// Mitsubishi GX Works2 project: BookEX6_42 DataControl   PLC: Q13UDV

// global labels: Global
VAR_GLOBAL
  bVar0 AT M5000 : BOOL;
  abArray0 AT M5010 : ARRAY [0..49] OF BOOL;
  sStr0 AT D5000 : STRING[199];
  sStr1 AT D5100 : STRING[199];
  sStr2 AT D5200 : STRING[199];
  sStr3 AT D5300 : STRING[199];
  sStr4 AT D5400 : STRING[199];
  sStr5 AT D5500 : STRING[199];
  sStr6 AT D5600 : STRING[199];
  sStr7 AT D5700 : STRING[199];
  sStr8 AT D5800 : STRING[199];
  sStr9 AT D5900 : STRING[199];
  iVar0 AT D4500 : INT;
  iVar1 AT D4501 : INT;
  iVar2 AT D4502 : INT;
  iVar3 AT D4503 : INT;
  iVar4 AT D4504 : INT;
  iVar5 AT D4505 : INT;
  iVar6 AT D4506 : INT;
  iVar7 AT D4507 : INT;
  iVar8 AT D4508 : INT;
  iVar9 AT D4509 : INT;
  dVar0 AT D4510 : DINT;
  dVar1 AT D4512 : DINT;
  dVar2 AT D4514 : DINT;
  dVar3 AT D4516 : DINT;
  dVar4 AT D4518 : DINT;
  dVar5 AT D4520 : DINT;
  dVar6 AT D4522 : DINT;
  dVar7 AT D4524 : DINT;
  dVar8 AT D4526 : DINT;
  dVar9 AT D4528 : DINT;
  wVar0 AT D4530 : WORD;
  wVar1 AT D4531 : WORD;
  wVar2 AT D4532 : WORD;
  wVar3 AT D4533 : WORD;
  wVar4 AT D4534 : WORD;
  wVar5 AT D4535 : WORD;
  wVar6 AT D4536 : WORD;
  wVar7 AT D4537 : WORD;
  wVar8 AT D4538 : WORD;
  wVar9 AT D4539 : WORD;
  dwVar0 AT D4540 : DWORD;
  dwVar1 AT D4542 : DWORD;
  dwVar2 AT D4544 : DWORD;
  dwVar3 AT D4546 : DWORD;
  dwVar4 AT D4548 : DWORD;
  dwVar5 AT D4550 : DWORD;
  dwVar6 AT D4552 : DWORD;
  dwVar7 AT D4554 : DWORD;
  dwVar8 AT D4556 : DWORD;
  dwVar9 AT D4558 : DWORD;
  fsVar0 AT D4560 : REAL;
  fsVar1 AT D4562 : REAL;
  fsVar2 AT D4564 : REAL;
  fsVar3 AT D4566 : REAL;
  fsVar4 AT D4568 : REAL;
  fsVar5 AT D4570 : REAL;
  fsVar6 AT D4572 : REAL;
  fsVar7 AT D4574 : REAL;
  fsVar8 AT D4576 : REAL;
  fsVar9 AT D4578 : REAL;
  fdVar0 AT D4580 : LREAL;
  tTime0 AT D4620 : TIME;
  tTime1 AT D4622 : TIME;
  tTime2 AT D4624 : TIME;
  tTime3 AT D4626 : TIME;
  tTime4 AT D4628 : TIME;
  tTime5 AT D4630 : TIME;
  tTime6 AT D4632 : TIME;
  tTime7 AT D4634 : TIME;
  tTime8 AT D4636 : TIME;
  tTime9 AT D4638 : TIME;
  tTime10 AT D4640 : TIME;
  bVar1 AT M5001 : BOOL;
  bVar2 AT M5002 : BOOL;
  bVar3 AT M5003 : BOOL;
  bVar4 AT M5004 : BOOL;
  bVar5 AT M5005 : BOOL;
  bVar6 AT M5006 : BOOL;
  bVar7 AT M5007 : BOOL;
  bVar8 AT M5008 : BOOL;
  bVar9 AT M5009 : BOOL;
  abArray1 AT M5060 : ARRAY [0..49] OF BOOL;
  abArray2 AT M5110 : ARRAY [0..49] OF BOOL;
  abArray3 AT M5160 : ARRAY [0..49] OF BOOL;
  abArray4 AT M5210 : ARRAY [0..49] OF BOOL;
  abArray5 AT M5260 : ARRAY [0..49] OF BOOL;
  abArray6 AT M5310 : ARRAY [0..49] OF BOOL;
  abArray7 AT M5360 : ARRAY [0..49] OF BOOL;
  abArray8 AT M5410 : ARRAY [0..49] OF BOOL;
  abArray9 AT M5460 : ARRAY [0..49] OF BOOL;
  fdVar1 AT D4584 : LREAL;
  fdVar2 AT D4588 : LREAL;
  fdVar3 AT D4592 : LREAL;
  fdVar4 AT D4596 : LREAL;
  fdVar5 AT D4600 : LREAL;
  fdVar6 AT D4604 : LREAL;
  fdVar7 AT D4608 : LREAL;
  fdVar8 AT D4612 : LREAL;
  fdVar9 AT D4616 : LREAL;
  afsPen0 AT D2000 : ARRAY [0..499] OF REAL;
  afsPen1 AT D3000 : ARRAY [0..499] OF REAL;
END_VAR
// user libraries (not included): HMI

FUNCTION realBAND
VAR_INPUT
  fs_Low : REAL;
  fs_High : REAL;
  fs_IN : REAL;
END_VAR
;
IF fs_IN < fs_Low THEN
	realBAND := fs_IN - fs_Low;
ELSIF fs_IN > fs_High THEN
	realBAND := fs_IN - fs_High;
ELSE
	realBAND := 0.0;
END_IF;
END_FUNCTION

FUNCTION realLIMIT
VAR_INPUT
  fs_Low : REAL;
  fs_High : REAL;
  fs_IN : REAL;
END_VAR
;
IF fs_IN < fs_Low THEN
	realLIMIT := fs_Low;
ELSIF fs_IN > fs_High THEN
	realLIMIT := fs_High;
ELSE
	realLIMIT := fs_IN;
END_IF;
END_FUNCTION

FUNCTION realSCL
VAR_INPUT
  i_Cnt : INT;
  afs_Data : ARRAY [0..19] OF REAL;
END_VAR
VAR
  ix : INT;
  iCnt : INT;
END_VAR
VAR_INPUT
  fs_InX : REAL;
END_VAR
VAR
  fs_OutY : REAL;
END_VAR
;
fs_OutY := fs_InX;
IF i_Cnt > 10 THEN iCnt := 9; ELSE iCnt := i_Cnt -1; END_IF;
FOR ix := 0 TO iCnt DO 
	IF fs_InX >=  afs_Data[ix*2] AND fs_InX < afs_Data[ix*2+2] THEN
		fs_OutY := afs_Data[ix*2+1] + (afs_Data[ix*2+3] - afs_Data[ix*2+1]) * (fs_InX - afs_Data[ix*2]) / (afs_Data[ix*2+2] - afs_Data[ix*2]); 
		EXIT;
	END_IF;
END_FOR;		
realSCL := fs_OutY;
END_FUNCTION

FUNCTION realZONE
VAR_INPUT
  fs_Low : REAL;
  fs_High : REAL;
  fs_IN : REAL;
END_VAR
;
IF fs_IN < 0.0 THEN
	realZONE := fs_IN + fs_Low;
ELSIF fs_IN > 0.0 THEN
	realZONE := fs_IN + fs_High;
ELSE
	realZONE := 0.0;
END_IF;
END_FUNCTION

PROGRAM ExBAND
VAR
  Mov4INT_1 : Mov4INT;
END_VAR
(* structured ladder/FBD written out as ST: instructions are called as NAME(EN, inputs, outputs); _pN, _eN, _tN stand for wires *)
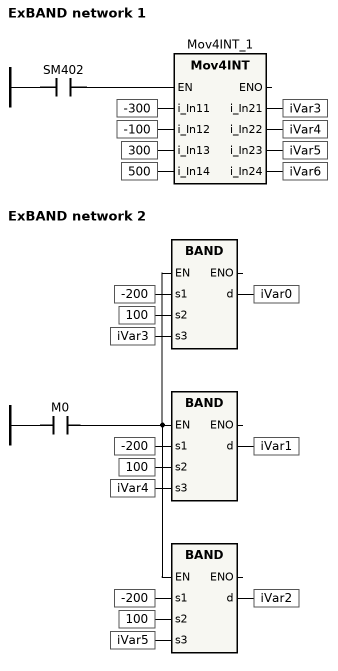
(* network 1 *)
Mov4INT_1(EN := SM402, i_In11 := -300, i_In12 := -100, i_In13 := 300, i_In14 := 500, i_In21 => iVar3, i_In22 => iVar4, i_In23 => iVar5, i_In24 => iVar6);
(* network 2 *)
BAND(M0, -200, 100, iVar3, iVar0);
BAND(M0, -200, 100, iVar4, iVar1);
BAND(M0, -200, 100, iVar5, iVar2);
END_PROGRAM

PROGRAM ExBAND_ST
VAR
  ix : INT;
  radx : REAL;
  fsx1 : REAL;
  fsx2 : REAL;
  fscale : REAL;
  fsIN : REAL;
END_VAR

fsVar8 := 1.0;
fsVar9 := -1.0;
 (* SIN *)
FOR ix := 0 TO 359 DO
	RAD(TRUE,INT_TO_REAL(ix),radx);
	SIN_E(TRUE, radx, fsx2);
	afsPen0[ix] := fsx2;
	afsPen1[ix] := realBAND(-0.2, 0.2, fsx2);
END_FOR;
END_PROGRAM

PROGRAM ExLIMIT
VAR
  Mov4INT_1 : Mov4INT;
END_VAR
(* structured ladder/FBD written out as ST: instructions are called as NAME(EN, inputs, outputs); _pN, _eN, _tN stand for wires *)
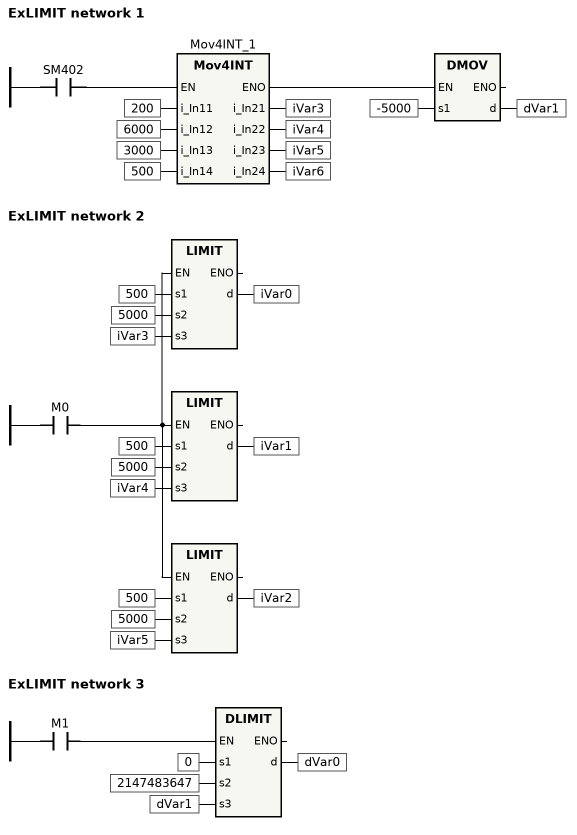
(* network 1 *)
Mov4INT_1(EN := SM402, i_In11 := 200, i_In12 := 6000, i_In13 := 3000, i_In14 := 500, i_In21 => iVar3, i_In22 => iVar4, i_In23 => iVar5, i_In24 => iVar6);
DMOV(Mov4INT_1.ENO, -5000, dVar1);
(* network 2 *)
LIMIT(M0, 500, 5000, iVar3, iVar0);
LIMIT(M0, 500, 5000, iVar4, iVar1);
LIMIT(M0, 500, 5000, iVar5, iVar2);
(* network 3 *)
DLIMIT(M1, 0, 2147483647, dVar1, dVar0);
END_PROGRAM

PROGRAM ExLIMIT_ST
VAR
  ix : INT;
  radx : REAL;
  fsx1 : REAL;
  fsx2 : REAL;
  fscale : REAL;
  fsIN : REAL;
END_VAR
fsVar8 := 1.0;
fsVar9 := -1.0;
 (* SIN *)
FOR ix := 0 TO 359 DO
	RAD(TRUE,INT_TO_REAL(ix),radx);
	SIN_E(TRUE, radx, fsx2);
	afsPen0[ix] := 0.0; (* fsx2; *)
	afsPen1[ix] := realLIMIT(-0.8, 0.8, fsx2);
END_FOR;
END_PROGRAM

PROGRAM ExSCL
VAR
  Mov8INT_1 : Mov8INT;
  Mov4INT_1 : Mov4INT;
  Mov8INT_2 : Mov8INT;
  Mov4INT_2 : Mov4INT;
  Mov8REAL_1 : Mov8REAL;
  Mov4REAL_1 : Mov4REAL;
  fsXY : ARRAY [0..19] OF REAL;
  fsX : REAL;
END_VAR
(* structured ladder/FBD written out as ST: instructions are called as NAME(EN, inputs, outputs); _pN, _eN, _tN stand for wires *)
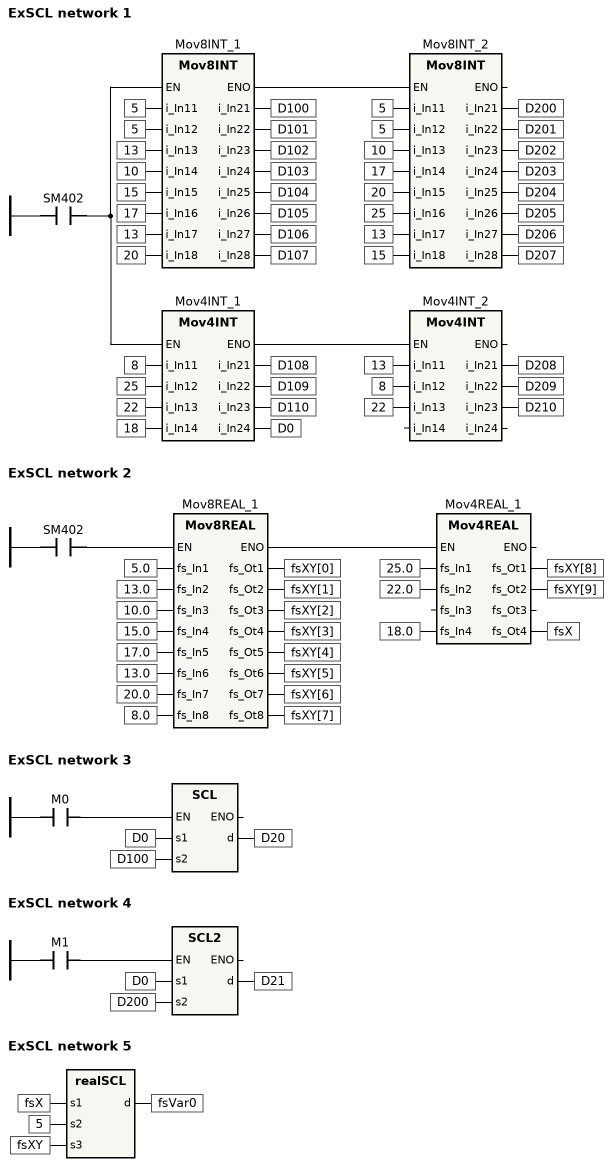
(* network 1 *)
Mov8INT_1(EN := SM402, i_In11 := 5, i_In12 := 5, i_In13 := 13, i_In14 := 10, i_In15 := 15, i_In16 := 17, i_In17 := 13, i_In18 := 20, i_In21 => D100, i_In22 => D101, i_In23 => D102, i_In24 => D103, i_In25 => D104, i_In26 => D105, i_In27 => D106, i_In28 => D107);
Mov8INT_2(EN := Mov8INT_1.ENO, i_In11 := 5, i_In12 := 5, i_In13 := 10, i_In14 := 17, i_In15 := 20, i_In16 := 25, i_In17 := 13, i_In18 := 15, i_In21 => D200, i_In22 => D201, i_In23 => D202, i_In24 => D203, i_In25 => D204, i_In26 => D205, i_In27 => D206, i_In28 => D207);
Mov4INT_1(EN := SM402, i_In11 := 8, i_In12 := 25, i_In13 := 22, i_In14 := 18, i_In21 => D108, i_In22 => D109, i_In23 => D110, i_In24 => D0);
Mov4INT_2(EN := Mov4INT_1.ENO, i_In11 := 13, i_In12 := 8, i_In13 := 22, i_In21 => D208, i_In22 => D209, i_In23 => D210);
(* network 2 *)
Mov8REAL_1(EN := SM402, fs_In1 := 5.0, fs_In2 := 13.0, fs_In3 := 10.0, fs_In4 := 15.0, fs_In5 := 17.0, fs_In6 := 13.0, fs_In7 := 20.0, fs_In8 := 8.0, fs_Ot1 => fsXY[0], fs_Ot2 => fsXY[1], fs_Ot3 => fsXY[2], fs_Ot4 => fsXY[3], fs_Ot5 => fsXY[4], fs_Ot6 => fsXY[5], fs_Ot7 => fsXY[6], fs_Ot8 => fsXY[7]);
Mov4REAL_1(EN := Mov8REAL_1.ENO, fs_In1 := 25.0, fs_In2 := 22.0, fs_In4 := 18.0, fs_Ot1 => fsXY[8], fs_Ot2 => fsXY[9], fs_Ot4 => fsX);
(* network 3 *)
SCL(M0, D0, D100, D20);
(* network 4 *)
SCL2(M1, D0, D200, D21);
(* network 5 *)
fsVar0 := realSCL(fsX, 5, fsXY);
END_PROGRAM

PROGRAM ExZONE
VAR
  Mov4INT_1 : Mov4INT;
END_VAR
(* structured ladder/FBD written out as ST: instructions are called as NAME(EN, inputs, outputs); _pN, _eN, _tN stand for wires *)
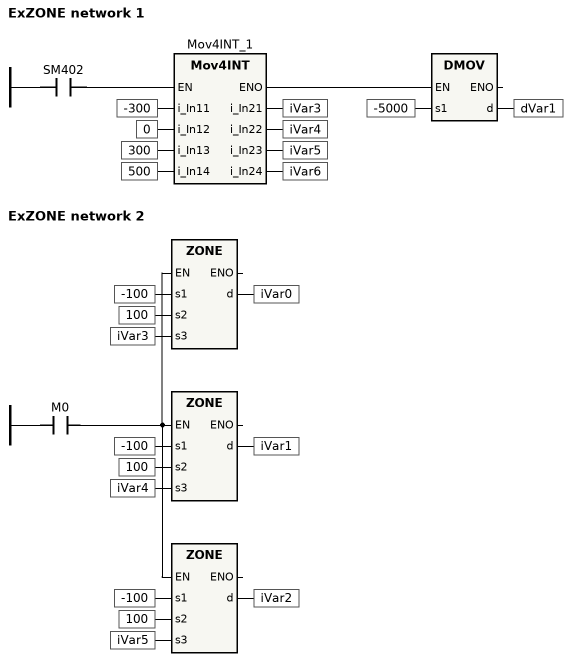
(* network 1 *)
Mov4INT_1(EN := SM402, i_In11 := -300, i_In12 := 0, i_In13 := 300, i_In14 := 500, i_In21 => iVar3, i_In22 => iVar4, i_In23 => iVar5, i_In24 => iVar6);
DMOV(Mov4INT_1.ENO, -5000, dVar1);
(* network 2 *)
ZONE(M0, -100, 100, iVar3, iVar0);
ZONE(M0, -100, 100, iVar4, iVar1);
ZONE(M0, -100, 100, iVar5, iVar2);
END_PROGRAM

PROGRAM ExZONE_ST
VAR
  ix : INT;
  radx : REAL;
  fsx1 : REAL;
  fsx2 : REAL;
  fscale : REAL;
  fsIN : REAL;
END_VAR
fsVar8 := 1.0;
fsVar9 := -1.0;
 (* SIN *)
FOR ix := 0 TO 359 DO
	RAD(TRUE,INT_TO_REAL(ix),radx);
	SIN_E(TRUE, radx, fsx2);
	fsIN := fsx2 * 0.9;
	afsPen0[ix] := fsIN;
	afsPen1[ix] := realZONE(-0.1, 0.1, fsIN);
END_FOR;
END_PROGRAM
